ABB RAPID module: Module1.mod

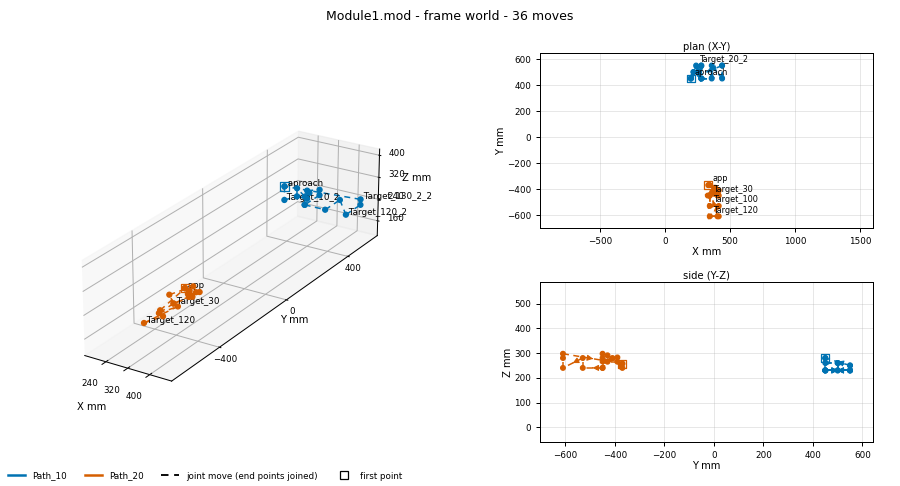
[picture p0: tool path of Module1.mod in frame world, 36 of 36 moves have a stored position in this frame; points joined in program order, loops and branches not executed]
MODULE Module1
    PERS wobjdata Grados:=[FALSE,TRUE,"",[[270,-370,200],[0.683012702,0.183012702,-0.183012702,-0.683012702]],[[0,0,-200],[1,0,0,0]]];
    TASK PERS wobjdata Workobject_2:=[FALSE,TRUE,"",[[0,0,0],[1,0,0,0]],[[0,0,0],[1,0,0,0]]];
    CONST robtarget Target_10_2:=[[200,450,230],[0,1,0,0],[0,2,0,1],[9E+09,9E+09,9E+09,9E+09,9E+09,9E+09]];
    CONST robtarget Target_20_2:=[[240,550,230],[0,1,0,0],[0,2,0,1],[9E+09,9E+09,9E+09,9E+09,9E+09,9E+09]];
    CONST robtarget Target_30_2:=[[280,450,230],[0,1,0,0],[0,2,0,1],[9E+09,9E+09,9E+09,9E+09,9E+09,9E+09]];
    CONST robtarget Target_40_2:=[[280,450,260],[0,1,0,0],[0,2,0,1],[9E+09,9E+09,9E+09,9E+09,9E+09,9E+09]];
    CONST robtarget Target_50_2:=[[220,500,230],[0,1,0,0],[0,2,0,1],[9E+09,9E+09,9E+09,9E+09,9E+09,9E+09]];
    CONST robtarget Target_60_2:=[[260,500,230],[0,1,0,0],[0,2,0,1],[9E+09,9E+09,9E+09,9E+09,9E+09,9E+09]];
    CONST robtarget Target_70_2:=[[260,500,260],[0,1,0,0],[0,2,0,1],[9E+09,9E+09,9E+09,9E+09,9E+09,9E+09]];
    CONST robtarget Target_80_2:=[[280,550,230],[0,1,0,0],[0,2,0,1],[9E+09,9E+09,9E+09,9E+09,9E+09,9E+09]];
    CONST robtarget Target_90_2:=[[280,450,230],[0,1,0,0],[0,2,0,1],[9E+09,9E+09,9E+09,9E+09,9E+09,9E+09]];
    CONST robtarget Target_100_2:=[[360,450,230],[0,1,0,0],[0,2,0,1],[9E+09,9E+09,9E+09,9E+09,9E+09,9E+09]];
    CONST robtarget Target_110_2:=[[360,550,230],[0,1,0,0],[0,2,0,1],[9E+09,9E+09,9E+09,9E+09,9E+09,9E+09]];
    CONST robtarget Target_120_2:=[[440,450,230],[0,1,0,0],[0,2,0,1],[9E+09,9E+09,9E+09,9E+09,9E+09,9E+09]];
    CONST robtarget Target_130_2:=[[440,550,230],[0,1,0,0],[0,2,0,1],[9E+09,9E+09,9E+09,9E+09,9E+09,9E+09]];
    CONST robtarget Target_10:=[[0,85.000000032,197.224318625],[0,-0.707106781,0.707106781,0],[-1,-2,0,1],[9E+09,9E+09,9E+09,9E+09,9E+09,9E+09]];
    CONST robtarget Target_20:=[[40,165.000000032,197.224318625],[0,-0.707106781,0.707106781,0],[-1,-2,0,1],[9E+09,9E+09,9E+09,9E+09,9E+09,9E+09]];
    CONST robtarget Target_30:=[[80,85.000000032,197.224318625],[0,-0.707106781,0.707106781,0],[-1,-2,0,1],[9E+09,9E+09,9E+09,9E+09,9E+09,9E+09]];
    CONST robtarget Target_40:=[[80,85.000000032,227.224318625],[0,-0.707106781,0.707106781,0],[-1,-2,0,1],[9E+09,9E+09,9E+09,9E+09,9E+09,9E+09]];
    CONST robtarget Target_50:=[[20,135.000000032,197.224318625],[0,-0.707106781,0.707106781,0],[-1,-2,0,1],[9E+09,9E+09,9E+09,9E+09,9E+09,9E+09]];
    CONST robtarget Target_60:=[[60,135.000000032,197.224318625],[0,-0.707106781,0.707106781,0],[-1,-2,0,1],[9E+09,9E+09,9E+09,9E+09,9E+09,9E+09]];
    CONST robtarget Target_70:=[[60,135.000000032,227.224318625],[0,-0.707106781,0.707106781,0],[-1,-2,0,1],[9E+09,9E+09,9E+09,9E+09,9E+09,9E+09]];
    CONST robtarget Target_80:=[[80,165.000000032,197.224318625],[0,-0.707106781,0.707106781,0],[-1,-2,0,1],[9E+09,9E+09,9E+09,9E+09,9E+09,9E+09]];
    CONST robtarget Target_90:=[[80,85.000000032,197.224318625],[0,-0.707106781,0.707106781,0],[-1,-2,0,1],[9E+09,9E+09,9E+09,9E+09,9E+09,9E+09]];
    CONST robtarget Target_100:=[[160,85.000000032,197.224318625],[0,-0.707106781,0.707106781,0],[-1,-2,0,1],[9E+09,9E+09,9E+09,9E+09,9E+09,9E+09]];
    CONST robtarget Target_110:=[[160,165.000000032,197.224318625],[0,-0.707106781,0.707106781,0],[-1,-2,0,1],[9E+09,9E+09,9E+09,9E+09,9E+09,9E+09]];
    CONST robtarget Target_120:=[[240,85.000000032,197.224318625],[0,-0.707106781,0.707106781,0],[-1,-2,0,1],[9E+09,9E+09,9E+09,9E+09,9E+09,9E+09]];
    CONST robtarget Target_130:=[[240,165.000000032,197.224318625],[0,-0.707106781,0.707106781,0],[-1,-2,0,1],[9E+09,9E+09,9E+09,9E+09,9E+09,9E+09]];
    TASK PERS wobjdata Wob:=[FALSE,TRUE,"",[[0,0,0],[1,0,0,0]],[[0,0,0],[1,0,0,0]]];
    CONST robtarget aproach:=[[200,450,280],[0,1,0,0],[0,2,0,1],[9E+09,9E+09,9E+09,9E+09,9E+09,9E+09]];
    CONST robtarget Target_80_2_2:=[[280,550,250],[0,1,0,0],[0,2,0,1],[9E+09,9E+09,9E+09,9E+09,9E+09,9E+09]];
    CONST robtarget Target_130_2_2:=[[440,550,250],[0,1,0,0],[0,2,0,1],[9E+09,9E+09,9E+09,9E+09,9E+09,9E+09]];
    CONST robtarget Target_50_2_2:=[[220,500,260],[0,1,0,0],[0,2,0,1],[9E+09,9E+09,9E+09,9E+09,9E+09,9E+09]];
    CONST robtarget app:=[[0,85.000000032,217.224318625],[0,-0.707106781,0.707106781,0],[-1,-2,0,1],[9E+09,9E+09,9E+09,9E+09,9E+09,9E+09]];
    CONST robtarget Target_50_4:=[[20,135.000000032,217.224318625],[0,-0.707106781,0.707106781,0],[-1,-2,0,1],[9E+09,9E+09,9E+09,9E+09,9E+09,9E+09]];
    CONST robtarget Target_130_3:=[[240,165.000000032,217.224318625],[0,-0.707106781,0.707106781,0],[-1,-2,1,1],[9E+09,9E+09,9E+09,9E+09,9E+09,9E+09]];
    CONST robtarget Target_80_3:=[[80,165.000000032,217.224318625],[0,-0.707106781,0.707106781,0],[-1,-2,0,1],[9E+09,9E+09,9E+09,9E+09,9E+09,9E+09]];
    PERS tooldata Marker:=[TRUE,[[-0.503,0,175.983],[1,0,0,0]],[0.12,[0.304,0,59.07],[1,0,0,0],0.001,0.001,0]];

!***********************************************************
    !
    ! Módulo:  Module1
    !
    ! Descripción:
    !   <Introduzca la descripción aquí>
    !
    ! Autor: USER
    !
    ! Versión: 1.0
    !
    !***********************************************************


    !***********************************************************
    !
    ! Procedimiento Main
    !
    !   Este es el punto de entrada de su programa
    !
    !***********************************************************
    PROC main()
        IF DI_01=1 THEN
            Path_10;
        ENDIF
        IF DI_02=1 THEN
            Path_20;
        ENDIF
    ENDPROC
    PROC Path_10()
        MoveJ aproach,v100,z10,tool0\WObj:=wob;
        MoveJ Target_10_2,v80,z10,tool0\WObj:=wob;
        MoveJ Target_20_2,v80,z10,tool0\WObj:=wob;
        MoveJ Target_30_2,v80,z10,tool0\WObj:=wob;
        MoveJ Target_40_2,v80,z10,tool0\WObj:=wob;
        MoveJ Target_50_2_2,v80,z10,tool0\WObj:=wob;
        MoveJ Target_50_2,v80,z10,tool0\WObj:=wob;
        MoveJ Target_60_2,v80,z10,tool0\WObj:=wob;
        MoveJ Target_70_2,v80,z10,tool0\WObj:=wob;
        MoveJ Target_80_2_2,v80,z10,tool0\WObj:=wob;
        MoveJ Target_80_2,v80,z10,tool0\WObj:=wob;
        MoveJ Target_90_2,v80,z10,tool0\WObj:=wob;
        MoveJ Target_100_2,v80,z10,tool0\WObj:=wob;
        MoveJ Target_110_2,v80,z10,tool0\WObj:=wob;
        MoveJ Target_120_2,v80,z10,tool0\WObj:=wob;
        MoveJ Target_130_2,v80,z10,tool0\WObj:=wob;
        MoveJ Target_130_2_2,v80,z10,tool0\WObj:=wob;
        MoveJ aproach,v100,z10,tool0\WObj:=wob;
    ENDPROC
    PROC Path_20()
        MoveJ app,v100,z10,tool0\WObj:=Grados;
        MoveJ Target_10,v80,z10,tool0\WObj:=Grados;
        MoveJ Target_20,v80,z10,tool0\WObj:=Grados;
        MoveJ Target_30,v80,z10,tool0\WObj:=Grados;
        MoveJ Target_40,v80,z10,tool0\WObj:=Grados;
        MoveJ Target_50_4,v80,z10,tool0\WObj:=Grados;
        MoveJ Target_50,v80,z10,tool0\WObj:=Grados;
        MoveJ Target_60,v80,z10,tool0\WObj:=Grados;
        MoveJ Target_70,v80,z10,tool0\WObj:=Grados;
        MoveJ Target_80_3,v80,z10,tool0\WObj:=Grados;
        MoveJ Target_80,v80,z10,tool0\WObj:=Grados;
        MoveJ Target_90,v80,z10,tool0\WObj:=Grados;
        MoveJ Target_100,v80,z10,tool0\WObj:=Grados;
        MoveJ Target_110,v80,z10,tool0\WObj:=Grados;
        MoveJ Target_120,v80,z10,tool0\WObj:=Grados;
        MoveJ Target_130,v80,z10,tool0\WObj:=Grados;
        MoveJ Target_130_3,v80,z10,tool0\WObj:=Grados;
        MoveJ app,v100,z10,tool0\WObj:=Grados;
    ENDPROC
ENDMODULE
